FUNCTION_BLOCK FB_HaltNC IMPLEMENTS I_Halt
VAR
    {attribute 'no_copy'}
    AxisRef : REFERENCE TO AXIS_REF;
    fbMcHalt 		: MC_Halt;
    sMessage : T_MAXSTRING;

END_VAR

IF NOT __ISVALIDREF(AxisRef) THEN
    RETURN;
END_IF

fbMcHalt(Axis := AxisRef );

PROPERTY Aborted : BOOL
GET
Aborted := THIS^.fbMcHalt.CommandAborted;
END_GET
END_PROPERTY

PROPERTY Active : BOOL
GET
Active := THIS^.fbMcHalt.Active;
END_GET
END_PROPERTY

PROPERTY Busy : BOOL
GET
Busy := THIS^.fbMcHalt.Busy;
END_GET
END_PROPERTY

METHOD PUBLIC CallAfterInit
VAR_INPUT
    AxisRef : REFERENCE TO AXIS_REF;
END_VAR
THIS^.AxisRef REF= AxisRef;
END_METHOD

PROPERTY CommandHalt : BOOL
SET
THIS^.fbMcHalt.Execute := CommandHalt;
END_SET
END_PROPERTY

PROPERTY Done : BOOL
GET
Done := THIS^.fbMcHalt.Done;
END_GET
END_PROPERTY

PROPERTY Error : BOOL
GET
Error := THIS^.fbMcHalt.Error;
END_GET
END_PROPERTY

PROPERTY ErrorID : UDINT
GET
ErrorID := THIS^.fbMcHalt.ErrorID;
END_GET
END_PROPERTY

//FB_Init is always available implicitly and it is used primarily for initialization.
//The return value is not evaluated. For a specific influence, you can also declare the
//methods explicitly and provide additional code there with the standard initialization
//code. You can evaluate the return value.
METHOD FB_Init: BOOL
VAR_INPUT
    bInitRetains: BOOL; // TRUE: the retain variables are initialized (reset warm / reset cold)
    bInCopyCode: BOOL;  // TRUE: the instance will be copied to the copy code afterward (online change)
    AxisRef : REFERENCE TO AXIS_REF;
END_VAR
THIS^.AxisRef REF= AxisRef;
END_METHOD

METHOD Halt
VAR_INPUT
    Deceleration	: LREAL := 0;
    Jerk	: LREAL := 0;
    BufferMode	: MC_BufferMode := MC_BufferMode.MC_Aborting;
END_VAR
// Clear previous status: MC_Halt auto clear this bit when Done is set.
fbMcHalt(Execute := FALSE,  Axis := THIS^.AxisRef);
// initiate a new halting request
fbMcHalt(Execute := TRUE,
    Axis := THIS^.AxisRef,
    Execute := TRUE,
    Deceleration := Deceleration,
    Jerk := Jerk,
    BufferMode := BufferMode);
END_METHOD

METHOD HaltDone
// Clear previous status: MC_Halt auto clear this bit when Done is set.
fbMcHalt(Execute := FALSE,  Axis := THIS^.AxisRef);
END_METHOD

PROPERTY Message : T_MAXSTRING
GET
Message  := sMessage;
END_GET
END_PROPERTY

END_FUNCTION_BLOCK

(* stored: Version 1.1.0.1
   POU FB_HaltNC: Id {c033f4f8-0634-4c06-a30f-6a4c2be036bc}, SpecialFunc None
   Property Aborted: Id {0a3b6722-2eb3-4ccd-aef0-1f467bbcc869}
   Get Get: Id {af5a55f0-647d-40ab-98bd-8c3f9ba0c756}
   Property Active: Id {04d62f93-14c5-45c5-834a-45619c35235a}
   Get Get: Id {4a5fb9e3-eee2-4c86-aac7-88671ef9bcae}
   Property Busy: Id {2883f0f4-4b95-4139-8a36-d2b2f3dcc31b}
   Get Get: Id {5b77bc7a-e864-4e13-ae17-e0016b7d86c8}
   Method CallAfterInit: Id {7068fa57-7e79-4554-a691-c8e89ace2f96}
   Property CommandHalt: Id {bbacc6b5-2150-42a2-9054-67af9aca1473}
   Set Set: Id {32dd52a4-4349-46b9-ad3d-b8776ebebd30}
   Property Done: Id {be7dfb74-7669-4f3f-93f0-cda14723d1f0}
   Get Get: Id {0f32e8ae-880b-42bd-b635-3e016d1c20ba}
   Property Error: Id {45d4ccdb-82f3-4b2c-ae9a-f7a118e27ac3}
   Get Get: Id {bbf7cb10-277f-4907-9b37-03e01cec3c96}
   Property ErrorID: Id {336845aa-0c0a-4c8a-b21e-bc9fafd47d20}
   Get Get: Id {d0994f69-d16e-4cfd-8b2d-204ea0c00d54}
   Method FB_Init: Id {18cebc01-b938-405d-8b68-4f57807b525a}
   Method Halt: Id {7d31f5d0-f1cb-401e-ae13-f0dc85da0693}
   Method HaltDone: Id {22a58216-660c-4b25-a8ed-e863b8c537cb}
   Property Message: Id {08e92b01-505f-4268-a83e-cb2252382ca8}
   Get Get: Id {8eca0745-b604-4b2a-98ba-3971c670c893} *)
